RoboDK station: Concept_3.rdk

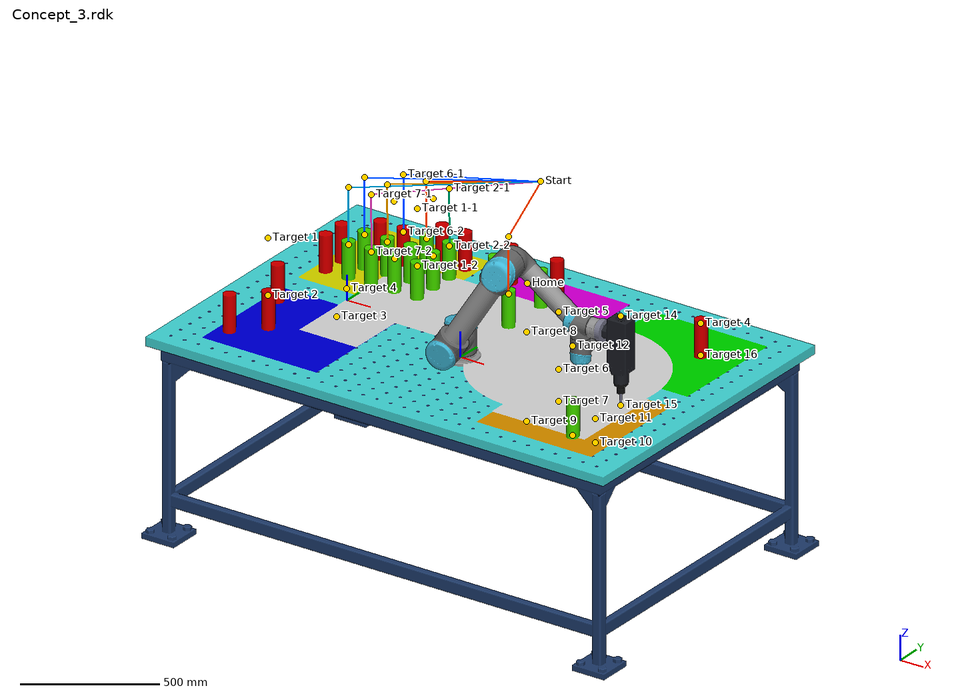
[picture v0: the station drawn from its stored meshes, robots at their saved joint values, targets as dots, program paths as lines]
Station Concept_3 (saved by RoboDK 5.3.4). Poses are relative to the parent item; angles as X-Y-Z fixed-axis rotations.
  - frame UR5 Base at (0, 0, 0) mm
    - robot UR5: 6 axes, payload 5 kg, reach 850 mm, repeatability 0.1 mm, weight 18.4 kg
        modified DH rows (alpha deg, a mm, theta deg, d mm): 0, 0, 0, 89.2; 90, 0, 180, 0; 0, 425, 0, 0; 0, 392.43, 0, 109; -90, 0, 0, 93.65; 90, 0, 180, 82
        joint limits [-360, -360, -360, -360, -360, -360] to [360, 360, 360, 360, 360, 360]; home [0, -90, -90, 0, 90, 0]; saved at [11.239, -121.743, -99.84, 41.507, 80.708, -269.961]
      - tool Spindle, TCP at (278.6, 0, 90) mm, rotated rx 0 ry 90 rz 0 deg, size 85 x 346.5 x 128 mm
  - frame Work Space at (-600, 150, 0) mm
    - object Cell Frame 3.5m at (0, 0, 0) mm, size 2018.1 x 1282.7 x 844.7 mm, geometry from Cell-Frame-3.5m.sld
    - object Table 2000x1200x800 at (0, 0, 0) mm, size 2020 x 1340 x 800 mm, geometry from Table-2000mmx1200mmx800mm.sld
  - frame Tubes at (0, 0, 0) mm
    - object Cylinder 1 at (0, 0, 0) mm, size 50 x 50 x 150 mm, geometry from Cylinder-100mmx300mm.sld
    - target Target 1-1 (Cartesian target) at (-400, 300, 360.05) mm, rotated rx -179.47 ry 0.1 rz 0.01 deg; joints [144.332, -85.591, -89.769, 355.486, 125.679, -270.457] of UR5
    - target Target 1-2 (Cartesian target) at (-400.41, 302.12, 131.43) mm, rotated rx -179.47 ry 0.1 rz 0.01 deg; joints [290.431, -87.073, 117.304, 149.477, -20.421, -270.256] of UR5
    - object Cylinder 2 at (0, 0, 0) mm, size 50 x 50 x 150 mm, geometry from Cylinder-100mmx300mm.sld
    - target Target 2-1 (Cartesian target) at (-400, 500, 360.05) mm, rotated rx -179.47 ry 0.1 rz 0.01 deg; joints [126.07, -110.39, -61.242, 351.805, 143.94, -270.39] of UR5
    - target Target 2-2 (Cartesian target) at (-400.41, 502.11, 131.43) mm, rotated rx -179.47 ry 0.1 rz 0.01 deg; joints [283.074, -64.973, 88.751, 155.77, -13.063, -270.09] of UR5
    - object Cylinder 3 at (0, 0, 0) mm, size 50 x 50 x 150 mm, geometry from Cylinder-100mmx300mm.sld
    - target Target 3-1 (Cartesian target) at (-400, 400, 360.05) mm, rotated rx -179.47 ry 0.1 rz 0.01 deg; joints [133.556, -97.311, -77.728, 355.187, 136.455, -270.423] of UR5
    - target Target 3-2 (Cartesian target) at (-400.41, 402.11, 131.43) mm, rotated rx -179.47 ry 0.1 rz 0.01 deg; joints [285.993, -76.138, 104.39, 151.377, -15.983, -270.173] of UR5
    - object Cylinder 4 at (0, 0, 0) mm, size 50 x 50 x 150 mm, geometry from Cylinder-100mmx300mm.sld
    - target Target 4-1 (Cartesian target) at (-500, 300, 360.05) mm, rotated rx -179.47 ry 0.1 rz 0.01 deg; joints [303.49, -84.873, 80.169, 184.519, -33.479, -270.376] of UR5
    - target Target 4-2 (Cartesian target) at (-500.41, 302.12, 131.43) mm, rotated rx -179.47 ry 0.1 rz 0.01 deg; joints [303.38, -78.184, 106.997, 151.001, -33.369, -270.375] of UR5
    - object Cylinder 5 at (0, 0, 0) mm, size 50 x 50 x 150 mm, geometry from Cylinder-100mmx300mm.sld
  - frame Zones at (0, 0, 0) mm
    - object Raw Material at (0, 0, 0) mm, size 500 x 500 x 0 mm, geometry from Square.sld
      - object Raw Material at (0, 0, 0) mm, size 500 x 500 x 0 mm, geometry from Square.sld
    - object Solution at (0, 0, 0) mm, size 500 x 500 x 0 mm, geometry from Square.sld
    - object Processing at (0, 0, 0) mm, size 500 x 500 x 0 mm, geometry from Square.sld
    - object Cleaning at (0, 0, 0) mm, size 500 x 500 x 0 mm, geometry from Square.sld
    - object Storage at (0, 0, 0) mm, size 500 x 500 x 0 mm, geometry from Square.sld
    - target Start (Cartesian target) at (0, 500, 500) mm, rotated rx -179.47 ry 0.1 rz 0.01 deg; joints [238.928, -64.181, 31.334, 213.045, 31.083, -270.699] of UR5
    - target Working prepare (Cartesian target) at (0, 500, 500) mm, rotated rx -179.47 ry 0.1 rz 0.01 deg; joints [238.928, -64.181, 31.334, 213.045, 31.083, -270.699] of UR5
    - target Home (Cartesian target) at (564.43, -387.6, 607.85) mm, rotated rx -90 ry 0 rz 180 deg; joints [0, -90, -90, 0, 90, 0] of UR5
    - target Target 4 (Cartesian target) at (700.11, 500.13, 131) mm, rotated rx 179.97 ry -0.07 rz -178.05 deg; joints [51.737, -139.979, -46.801, 6.665, 40.211, -269.885] of UR5
  - frame Room test at (0, 0, 0) mm
    - object Test 5 at (0, 0, 0) mm, size 50 x 50 x 150 mm, geometry from Cylinder-100mmx300mm.sld
    - target Target 5-1 (Cartesian target) at (-500, 500, 360.05) mm, rotated rx -179.47 ry 0.1 rz 0.01 deg; joints [292.814, -61.605, 49.602, 191.74, -22.803, -270.287] of UR5
    - target Target 5-2 (Cartesian target) at (-500.41, 502.11, 131.43) mm, rotated rx -179.47 ry 0.1 rz 0.01 deg; joints [292.771, -58.806, 79.19, 159.352, -22.76, -270.287] of UR5
    - object Test 6 at (0, 0, 0) mm, size 50 x 50 x 150 mm, geometry from Cylinder-100mmx300mm.sld
    - target Target 6-1 (Cartesian target) at (-600.41, 502.11, 360) mm, rotated rx -179.47 ry 0.1 rz 0.01 deg; joints [301.044, -48.579, 28.187, 200.194, -31.033, -270.36] of UR5
    - target Target 6-2 (Cartesian target) at (-600.41, 502.12, 131.43) mm, rotated rx -179.47 ry 0.1 rz 0.01 deg; joints [301.044, -50.573, 65.551, 164.824, -31.033, -270.36] of UR5
    - object Test 7 at (0, 0, 0) mm, size 50 x 50 x 150 mm, geometry from Cylinder-100mmx300mm.sld
    - target Target 7-1 (Cartesian target) at (-600, 300, 360.05) mm, rotated rx -179.47 ry 0.1 rz 0.01 deg; joints [313.089, -73.599, 66.605, 186.844, -43.079, -270.421] of UR5
    - target Target 7-2 (Cartesian target) at (-600.41, 302.12, 131.43) mm, rotated rx -179.47 ry 0.1 rz 0.01 deg; joints [312.961, -68.384, 93.771, 154.463, -42.95, -270.42] of UR5
    - object Test 8 at (0, 0, 0) mm, size 50 x 50 x 150 mm, geometry from Cylinder-100mmx300mm.sld
    - target Target 8-1 (Cartesian target) at (-600, 400, 360.05) mm, rotated rx -179.47 ry 0.1 rz 0.01 deg; joints [306.324, -63.678, 52.727, 190.778, -36.313, -270.391] of UR5
    - target Target 8-2 (Cartesian target) at (-600.41, 402.12, 131.43) mm, rotated rx -179.47 ry 0.1 rz 0.01 deg; joints [306.232, -60.399, 81.718, 158.508, -36.221, -270.391] of UR5
    - object Test 9 at (0, 0, 0) mm, size 50 x 50 x 150 mm, geometry from Cylinder-100mmx300mm.sld
    - object Test 10 at (0, 0, 0) mm, size 50 x 50 x 150 mm, geometry from Cylinder-100mmx300mm.sld
    - object Test 11 at (0, 0, 0) mm, size 50 x 50 x 150 mm, geometry from Cylinder-100mmx300mm.sld
    - target Target 11-1 (Cartesian target) at (-700, 300, 360.05) mm, rotated rx -179.47 ry 0.1 rz 0.01 deg; joints [320.212, -59.848, 46.891, 192.824, -50.202, -270.445] of UR5
    - target Target 11-2 (Cartesian target) at (-700.41, 302.12, 131.43) mm, rotated rx -179.47 ry 0.1 rz 0.01 deg; joints [320.082, -57.595, 77.244, 160.218, -50.071, -270.444] of UR5
    - object Test 12 at (0, 0, 0) mm, size 50 x 50 x 150 mm, geometry from Cylinder-100mmx300mm.sld
    - target Target 12-1 (Cartesian target) at (-700, 400, 360.05) mm, rotated rx -179.47 ry 0.1 rz 0.01 deg; joints [313.504, -47.85, 26.888, 200.814, -43.494, -270.422] of UR5
    - target Target 12-2 (Cartesian target) at (-700.41, 402.12, 131.43) mm, rotated rx -179.47 ry 0.1 rz 0.01 deg; joints [313.402, -49.958, 64.496, 165.313, -43.392, -270.422] of UR5
    - object Test 13 at (0, 0, 0) mm, size 50 x 50 x 150 mm, geometry from Cylinder-100mmx300mm.sld
    - object Test 14 at (0, 0, 0) mm, size 50 x 50 x 150 mm, geometry from Cylinder-100mmx300mm.sld
    - object Test 15 at (0, 0, 0) mm, size 50 x 50 x 150 mm, geometry from Cylinder-100mmx300mm.sld
    - object Test 16 at (0, 0, 0) mm, size 50 x 50 x 150 mm, geometry from Cylinder-100mmx300mm.sld
    - object Test 17 at (0, 0, 0) mm, size 50 x 50 x 150 mm, geometry from Cylinder-100mmx300mm.sld
    - object Test 18 at (0, 0, 0) mm, size 50 x 50 x 150 mm, geometry from Cylinder-100mmx300mm.sld
    - target Target 18-1 (Cartesian target) at (0, 300, 360) mm, rotated rx -179.47 ry 0.1 rz 0.01 deg; joints [221.409, -98.788, 93.609, 185.315, 48.602, -270.62] of UR5
    - target Target 18-2 (Cartesian target) at (0, 300, 131) mm, rotated rx -179.47 ry 0.1 rz 0.01 deg; joints [221.409, -91.712, 122.078, 149.771, 48.602, -270.62] of UR5
    - object Test 19 at (0, 0, 0) mm, size 50 x 50 x 150 mm, geometry from Cylinder-100mmx300mm.sld
    - object Test 20 at (0, 0, 0) mm, size 50 x 50 x 150 mm, geometry from Cylinder-100mmx300mm.sld
  - program Test tube 6 (8 instructions, listed below)
  - program Test tube 5 (8 instructions, listed below)
  - program Test tube 2 (8 instructions, listed below)
  - program Test tube 7 (8 instructions, listed below)
  - program Back home (4 instructions, listed below)
  - program Test tube 8 (8 instructions, listed below)
  - program Test tube 11 (8 instructions, listed below)
  - program Test tube 12 (8 instructions, listed below)
  - program Test tube 18 (9 instructions, listed below)
  - frame Room test 2 at (0, 0, 0) mm
    - object Test 21 at (0, 0, 0) mm, size 50 x 50 x 150 mm, geometry from Cylinder-100mmx300mm.sld
    - object Test 22 at (0, 0, 0) mm, size 50 x 50 x 150 mm, geometry from Cylinder-100mmx300mm.sld
    - object Test 23 at (0, 0, 0) mm, size 50 x 50 x 150 mm, geometry from Cylinder-100mmx300mm.sld
    - object Test 24 at (0, 0, 0) mm, size 50 x 50 x 150 mm, geometry from Cylinder-100mmx300mm.sld
    - object Test 25 at (0, 0, 0) mm, size 50 x 50 x 150 mm, geometry from Cylinder-100mmx300mm.sld
    - target Target 1 (Cartesian target) at (-700, -200, 360) mm, rotated rx -179.47 ry 0.1 rz 0.01 deg; joints [212.127, -113.227, -57.258, 350.605, 57.883, -270.594] of UR5
    - target Target 2 (Cartesian target) at (-700, -200, 131) mm, rotated rx -179.47 ry 0.1 rz 0.01 deg; joints [212.127, -198.585, 85.828, 292.877, 57.883, -270.594] of UR5
    - target Target 3 (Cartesian target) at (-400, -200, 131) mm, rotated rx -179.47 ry 0.1 rz 0.01 deg; joints [242.646, -200.573, -232.676, 253.472, 27.365, -270.727] of UR5
    - target Target 4 (Cartesian target) at (-500.74, 4.21, 131) mm, rotated rx -179.47 ry 0.1 rz 0.01 deg; joints [340.315, -93.95, 124.177, 149.665, -70.304, -270.493] of UR5
    - target Target 5 (Cartesian target) at (500.11, -100.13, 360) mm, rotated rx 179.97 ry -0.07 rz -178.05 deg; joints [0.508, -81.435, -93.344, -5.296, 91.44, -269.975] of UR5
    - target Target 6 (Cartesian target) at (500.11, -100.13, 131) mm, rotated rx 179.97 ry -0.07 rz -178.05 deg; joints [0.508, -88.465, -121.815, 30.205, 91.44, -269.975] of UR5
    - target Target 7 (Cartesian target) at (500.11, -100.13, 5) mm, rotated rx 179.97 ry -0.07 rz -178.05 deg; joints [0.508, -102.508, -130.621, 53.055, 91.44, -269.975] of UR5
    - target Target 8 (Cartesian target) at (500.11, -300.13, 360) mm, rotated rx 179.97 ry -0.07 rz -178.05 deg; joints [-28.923, -96.007, -79.124, -4.956, 120.871, -270.018] of UR5
    - target Target 9 (Cartesian target) at (500.11, -300.13, 5) mm, rotated rx 179.97 ry -0.07 rz -178.05 deg; joints [-28.923, -113.53, -113.832, 47.275, 120.871, -270.018] of UR5
    - target Target 10 (Cartesian target) at (800.11, -300.13, 5) mm, rotated rx 179.97 ry -0.07 rz -178.05 deg; joints [-16.995, -141.659, -62.83, 24.41, 108.943, -269.999] of UR5
    - target Target 11 (Cartesian target) at (800.11, -300.13, 100) mm, rotated rx 179.97 ry -0.07 rz -178.05 deg; joints [-16.995, -136.783, -57.234, 13.938, 108.943, -269.999] of UR5
    - target Target 12 (Cartesian target) at (700.11, -300.13, 360) mm, rotated rx 179.97 ry -0.07 rz -178.05 deg; joints [-19.795, -121.076, -45.37, -13.634, 111.743, -270.003] of UR5
    - target Target 13 (Cartesian target) at (700.11, -300.13, 5) mm, rotated rx 179.97 ry -0.07 rz -178.05 deg; joints [-19.795, -130.656, -83.697, 34.273, 111.743, -270.003] of UR5
    - target Target 14 (Cartesian target) at (700.11, -0.13, 360) mm, rotated rx 179.97 ry -0.07 rz -178.05 deg; joints [11.239, -107.527, -65.049, -7.499, 80.708, -269.961] of UR5
    - target Target 15 (Cartesian target) at (700.11, -0.13, 5) mm, rotated rx 179.97 ry -0.07 rz -178.05 deg; joints [11.239, -121.743, -99.84, 41.507, 80.708, -269.961] of UR5
    - target Target 16 (Cartesian target) at (700.11, 500.13, 5) mm, rotated rx 179.97 ry -0.07 rz -178.05 deg; joints [51.737, -145.225, -55.899, 21.008, 40.211, -269.885] of UR5
  - frame Working area at (0, 0, 0) mm
    - object Square at (0, 0, 3) mm, size 405 x 405 x 0 mm, geometry from Square.sld
      - object Circle at (0, 0, 0) mm, size 750 x 750 x 0 mm, geometry from Circle.sld
    - object Square at (0, 0, 0) mm, size 427.5 x 427.5 x 0 mm, geometry from Square.sld
    - object Square at (0, 0, 0) mm, size 427.5 x 427.5 x 0 mm, geometry from Square.sld
    - object Square at (0, 0, 0) mm, size 427.5 x 427.5 x 0 mm, geometry from Square.sld
    - object Square at (0, 0, 2) mm, size 250 x 250 x 0 mm, geometry from Square.sld
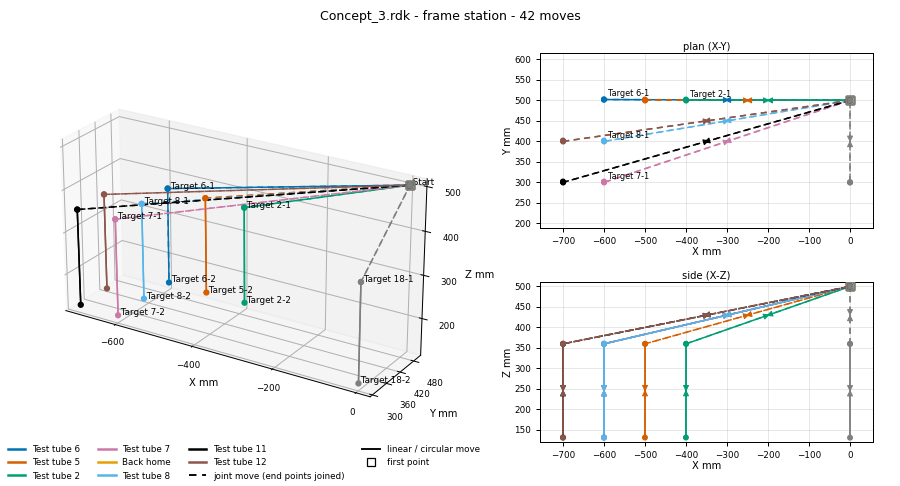
[picture p0: tool path of Concept_3.rdk in frame station, 42 of 42 moves have a stored position in this frame; points joined in program order, loops and branches not executed]

--- program Test tube 6 (robot UR5) ---
  替换物体
  设置参考: Zones
  设置工具: Spindle
  MoveL (Start)
  MoveJ (Target 6-1)
  MoveJ (Target 6-2)
  MoveL (Target 6-1)
  MoveL (Working prepare)

--- program Test tube 5 (robot UR5) ---
  替换物体
  设置参考: Zones
  设置工具: Spindle
  MoveJ (Start)
  MoveJ (Target 5-1)
  MoveL (Target 5-2)
  MoveL (Target 5-1)
  MoveJ (Working prepare)

--- program Test tube 2 (robot UR5) ---
  替换物体
  设置参考: Zones
  设置工具: Spindle
  MoveJ (Start)
  MoveL (Target 2-1)
  MoveL (Target 2-2)
  MoveL (Target 2-1)
  MoveJ (Working prepare)

--- program Test tube 7 (robot UR5) ---
  替换物体
  设置参考: Zones
  设置工具: Spindle
  MoveJ (Start)
  MoveJ (Target 7-1)
  MoveL (Target 7-2)
  MoveL (Target 7-1)
  MoveJ (Working prepare)

--- program Back home (robot UR5) ---
  替换物体
  设置参考: Zones
  设置工具: Spindle
  MoveJ (Start)

--- program Test tube 8 (robot UR5) ---
  替换物体
  设置参考: Zones
  设置工具: Spindle
  MoveJ (Start)
  MoveJ (Target 8-1)
  MoveL (Target 8-2)
  MoveL (Target 8-1)
  MoveJ (Working prepare)

--- program Test tube 11 (robot UR5) ---
  替换物体
  设置参考: Zones
  设置工具: Spindle
  MoveJ (Start)
  MoveJ (Target 11-1)
  MoveL (Target 11-2)
  MoveL (Target 11-1)
  MoveJ (Working prepare)

--- program Test tube 12 (robot UR5) ---
  替换物体
  设置参考: Zones
  设置工具: Spindle
  MoveJ (Start)
  MoveJ (Target 12-1)
  MoveL (Target 12-2)
  MoveL (Target 12-1)
  MoveJ (Working prepare)

--- program Test tube 18 (robot UR5) ---
  替换物体
  设置参考: Zones
  设置工具: Spindle
  MoveJ (Start)
  MoveJ (Working prepare)
  MoveJ (Target 18-1)
  MoveL (Target 18-2)
  MoveL (Target 18-1)
  MoveJ (Working prepare)
